{attribute 'qualified_only'}
{attribute 'strict'}
TYPE E_ModuleSequenceCommand :
(
	Enable,
	Disable,
	Start,
	Resume,
	Reset,
	Clear	
);
END_TYPE

(* stored: Version 1.1.0.1, ProductVersion 3.1.4024.9
   DUT E_ModuleSequenceCommand: Id {eb3d6b49-adde-47fa-9770-5fb2e21c491d} *)
